(* CoDeSys 2.3 export: CALLBACKNETVAR.EXP *)

(* POU NetVar POUs/CallbackNetVar, ST *)
FUNCTION CallbackNetVar:BYTE
VAR_INPUT
	dwEvent			: DWORD;
	dwFilter		: DWORD;
	dwOwner			: DWORD;
END_VAR
(* @TEXT_IMPLEMENTATION := 'ST' *)
IF (dwEvent = EVENT_STOP OR dwEvent = EVENT_BEFORE_RESET OR dwEvent = EVENT_BEFORE_DOWNLOAD) THEN
	NetVarManager_Udp.CloseSockets();
END_IF

IF (dwEvent = EVENT_DEBUG_LOOP) THEN
	(* Call die NetVarManager_Udp for Flush the Socket-Buffer while
		a BreakPoint is Activ in the IEC-Programm *)
	NetVarManager_Udp();
END_IF
END_FUNCTION
